FUNCTION_BLOCK FB_Sunblind
VAR_INPUT
	nFassade 			: INT;
	bPraesenz_Nachlauf	: BOOL;
	bTaster_Up			: BOOL;
	bTaster_Down		: BOOL;
	bSetPos				: BOOL;
	nPosValue			: INT;
	bSetAngl			: BOOL;
	nAnglValue			: INT;
	bEnable_SunPrtc_Thermo: BOOL;
	bEMA_Mode			: BOOL;
	rTemp_Ist				: REAL;
	rTemp_Soll				: REAL;
	rTemp_Hys				: REAL;
END_VAR

VAR_OUTPUT
	bRaff_Up			: BOOL;
	bRaff_Down			: BOOL;
	lrRaff_Pos			: LREAL;
	lrRaff_Angle		: LREAL;
	sModus				: STRING;
	bRaff_ManMod		: BOOL;
END_VAR
VAR
	FB_BA_SunPrtc 			: FB_BA_SunPrtc;
	FB_BA_SunBldWthrPrtc 	: FB_BA_SunBldWthrPrtc;
	FB_BA_SunBldPrioSwi8	: FB_BA_SunBldPrioSwi8;
	FB_ManSwitch			: FB_ManSwitch;
	FB_Abgleich_Raff		: FB_Abgleich_Raff;
	FB_EB_SunBldSwi			: FB_EB_SunBldSwi;
	FB_BA_SunBldActr		: FB_BA_SunBldActr;
	FB_BA_BrtnsHysDly		: FB_BA_BrtnsHysDly;
	FB_EMA					: FB_EMA;
	FB_Thermo				: FB_Thermo;
	FB_FassadenCheck		: FB_FassadenCheck;
	FB_Prio_Auswertung		: FB_Prio_Auswertung;
	
	nRaffPos				: INT;
	nRaffAngl				: INT;
	bClicked				: BOOL;
	FB_Set_Value			: FB_Set_Value;
	
	TON_Man					: TON;
	FB_LIGHT_Man			: FB_LIGHT;
	TP_Up					: TP;
	TP_Down					: TP;
	F_TRIG					: F_TRIG;
END_VAR
VAR // added by the converter: edge detectors and wires of the graphical bodies
    _w1, _w2 : BOOL;
END_VAR

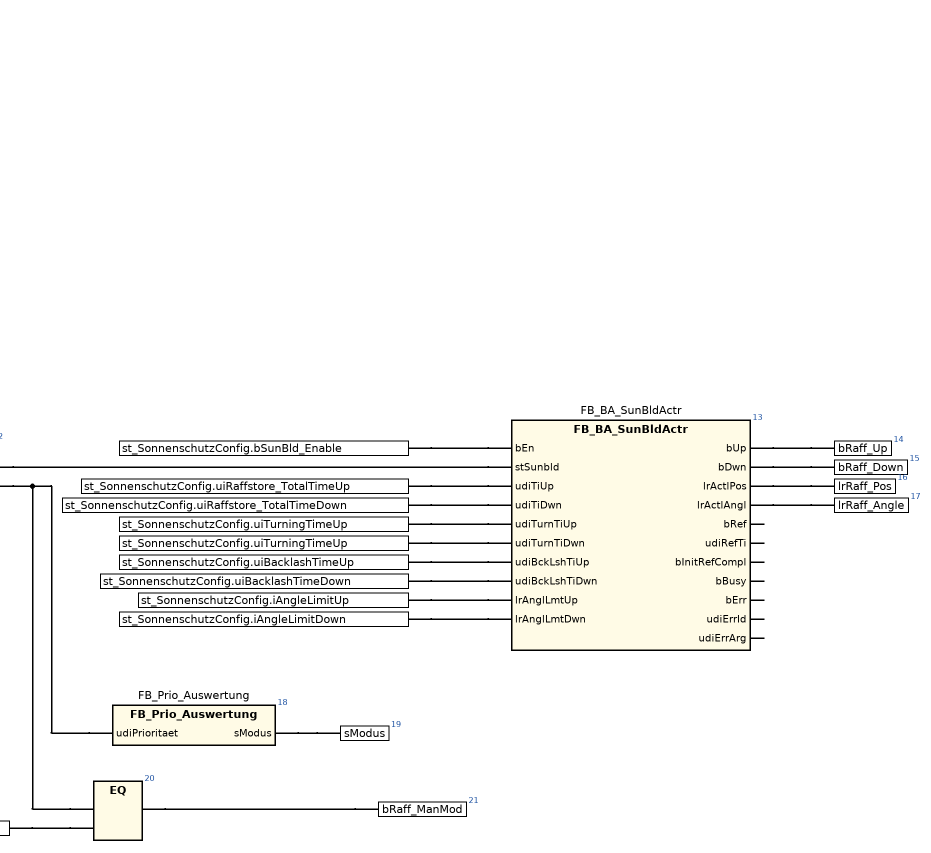
_w1 := bTaster_Up OR bRaff_Zentral_EMA_Auf;
_w2 := bTaster_Down OR bRaff_Zentral_Runter;
FB_EMA(bEMA := bEMA_Scharf AND bEMA_Mode);
F_TRIG(CLK := bRaffstore_Sperrung);
FB_ManSwitch(
    bTaster_Up := _w1,
    bTaster_Down := _w2,
    bSlider_Clicked := bClicked,
    bReset := F_TRIG.Q OR bRaff_Zentral_Reset);
FB_Abgleich_Raff(
    lrActualPos := FB_BA_SunBldActr.lrActlPos,
    lrActualAngle := FB_BA_SunBldActr.lrActlAngl,
    st_SunBld_Stellwert := FB_BA_SunBldPrioSwi8.stSunBld,
    nRaff_Pos := nRaffPos,
    nRaff_Angle := nRaffAngl);
FB_EB_SunBldSwi(
    bEn := FB_ManSwitch.bManMod_Enable,
    bUp := FB_ManSwitch.bRaff_Up,
    bDwn := FB_ManSwitch.bRaff_Down,
    bPos_steht := FB_Abgleich_Raff.bPos_steht,
    bSet_Angle := FB_Abgleich_Raff.bSet_Angle,
    bClicked := bClicked,
    nSlid_Pos := nRaffPos,
    nSlid_Angl := nRaffAngl,
    uiSwiOvrTi := st_SonnenschutzConfig.ui_SwitchOverTime);
FB_FassadenCheck(nFassade := nFassade);
FB_Thermo(
    bEnable := FB_FassadenCheck.bSunBld_Enable AND st_SonnenschutzConfig.bThermoautomatik_Enable AND bEnable_SunPrtc_Thermo,
    nFassade := nFassade,
    rTemperatur_Ist := rTemp_Ist,
    rTemperatur_Soll := rTemp_Soll,
    rHysterese := rTemp_Hys);
FB_BA_SunBldPrioSwi8(
    stSunBld_Prio1 := FB_Raffstore_Global.FB_BA_SunBldWthrPrtc.stSunbld,
    stSunBld_Prio2 := FB_EMA.ST_BA_SunBld,
    stSunBld_Prio3 := FB_EB_SunBldSwi.st_SunBld,
    stSunBld_Prio4 := FB_Thermo.ST_BA_SunBld);
FB_BA_SunBldActr(
    bEn := st_SonnenschutzConfig.bSunBld_Enable,
    stSunbld := FB_BA_SunBldPrioSwi8.stSunbld,
    udiTiUp := st_SonnenschutzConfig.uiRaffstore_TotalTimeUp,
    udiTiDwn := st_SonnenschutzConfig.uiRaffstore_TotalTimeDown,
    udiTurnTiUp := st_SonnenschutzConfig.uiTurningTimeUp,
    udiTurnTiDwn := st_SonnenschutzConfig.uiTurningTimeUp,
    udiBckLshTiUp := st_SonnenschutzConfig.uiBacklashTimeUp,
    udiBckLshTiDwn := st_SonnenschutzConfig.uiBacklashTimeDown,
    lrAnglLmtUp := st_SonnenschutzConfig.iAngleLimitUp,
    lrAnglLmtDwn := st_SonnenschutzConfig.iAngleLimitDown);
bRaff_Up := FB_BA_SunBldActr.bUp;
bRaff_Down := FB_BA_SunBldActr.bDwn;
lrRaff_Pos := FB_BA_SunBldActr.lrActlPos;
lrRaff_Angle := FB_BA_SunBldActr.lrActlAngl;
FB_Prio_Auswertung(udiPrioritaet := FB_BA_SunBldPrioSwi8.udiActvPrio);
sModus := FB_Prio_Auswertung.sModus;
bRaff_ManMod := FB_BA_SunBldPrioSwi8.udiActvPrio = 3;
FB_Set_Value(
    bSetPos := bSetPos,
    nPosValue := nPosValue,
    bSetAngl := bSetAngl,
    nAnglValue := nAnglValue,
    nRaff_Pos := nRaffPos,
    nRaff_Angle := nRaffAngl,
    bClicked := bClicked);

END_FUNCTION_BLOCK

(* stored: Version 1.1.0.1, ProductVersion 3.1.4024.12
   POU FB_Sunblind: Id {90aca38b-3e07-48fc-b761-c878e53b42d2}, SpecialFunc None *)
